{attribute 'qualified_only'}
VAR_GLOBAL CONSTANT
	DEG_TO_RAD : LREAL := PI/180.0;
	RAD_TO_DEG : LREAL := 180.0/PI;
	GEAR_RATIO : ARRAY [0..2] OF UINT := [61, 50, 35];
END_VAR

(* stored: Version 1.1.0.1, ProductVersion 3.1.4024.9
   GVL CONSTANTS: Id {30160ff0-ea78-4fb0-89e7-23814721b7a0} *)
